FUNCTION_BLOCK E_DELAY_V_D_ZERO (* Composite Function Block Type *)
  (* Standard: 61499-2 *)
  (* Version 0.0, 2/4/2026, SESA713705, Schneider Electric, template *)
  PACKAGE SE.Nereda;
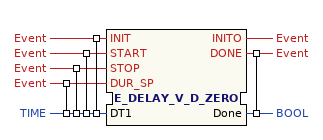
  EVENT_INPUT
    INIT WITH DT1;
    START WITH DT1; (* Begin Delay *)
    STOP WITH DT1; (* Cancel Delay *)
    DUR_SP WITH DT1;
  END_EVENT
  EVENT_OUTPUT
    INITO;
    DONE WITH Done; (* Input changed *)
  END_EVENT
  VAR_INPUT
    DT1 : TIME; (* Delay Time *)
  END_VAR
  VAR_OUTPUT
    Done : BOOL; (* Output value *)
  END_VAR
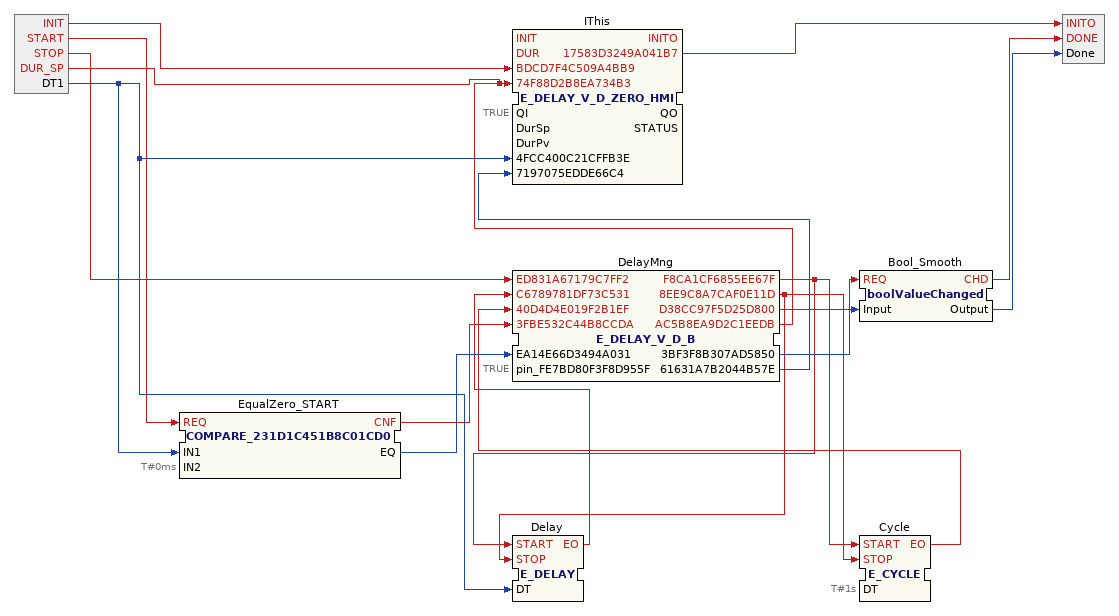
  FBS
    Bool_Smooth : boolValueChanged;
    IThis : E_DELAY_V_D_ZERO_HMI(QI := TRUE);
    DelayMng : E_DELAY_V_D_B(pin_FE7BD80F3F8D955F := TRUE);
    Delay : E_DELAY;
    Cycle : E_CYCLE(DT := T#1s);
    EqualZero_START : COMPARE_231D1C451B8C01CD0(IN2 := T#0ms); {SET_ATTRIBUTE(Configuration.GenericFBType.InterfaceParams, Runtime.Standard#CNT:=2;IN${CNT$}:TIME)}
  END_FBS
  EVENT_CONNECTIONS
    Bool_Smooth.CHD TO DONE;
    STOP TO DelayMng.ED831A67179C7FF2;
    Delay.EO TO DelayMng.C6789781DF73C531;
    Cycle.EO TO DelayMng.40D4D4E019F2B1EF;
    DelayMng.F8CA1CF6855EE67F TO Delay.START;
    DelayMng.F8CA1CF6855EE67F TO Cycle.START;
    DelayMng.8EE9C8A7CAF0E11D TO Delay.STOP;
    DelayMng.8EE9C8A7CAF0E11D TO Cycle.STOP;
    DelayMng.D38CC97F5D25D800 TO Bool_Smooth.REQ;
    START TO EqualZero_START.REQ;
    EqualZero_START.CNF TO DelayMng.3FBE532C44B8CCDA;
    INIT TO IThis.BDCD7F4C509A4BB9;
    DelayMng.AC5B8EA9D2C1EEDB TO IThis.74F88D2B8EA734B3;
    DUR_SP TO IThis.74F88D2B8EA734B3;
    IThis.17583D3249A041B7 TO INITO;
  END_CONNECTIONS
  DATA_CONNECTIONS
    Bool_Smooth.Output TO Done;
    DT1 TO Delay.DT;
    DelayMng.3BF3F8B307AD5850 TO Bool_Smooth.Input;
    DT1 TO EqualZero_START.IN1;
    EqualZero_START.EQ TO DelayMng.EA14E66D3494A031;
    DT1 TO IThis.4FCC400C21CFFB3E;
    DelayMng.61631A7B2044B57E TO IThis.7197075EDDE66C4;
  END_CONNECTIONS
END_FUNCTION_BLOCK
